// TIA Portal V16 export
// export: Created 2022-02-04T14:40:11.8651462Z, ExportSetting WithDefaults, DisplayName Totally Integrated Automation Portal, DisplayVersion V16 Update 1, DisplayName TIA Portal Version Control Interface, DisplayVersion V16, DisplayName TIA Portal Openness, DisplayVersion V16, DisplayName SINAMICS Startdrive Advanced, DisplayVersion V16 Update 5, DisplayName SINAMICS Startdrive G130, G150, S120, S150, SINAMICS MV, S210, DisplayVersion V16 Update 5, DisplayName SINAMICS Startdrive G110M, G120, G120C, G120D, G120P, G115D, DisplayVersion V16 Update 5, DisplayName STEP 7 Professional, DisplayVersion V16, DisplayName STEP 7 Safety, DisplayVersion V16, DisplayName WinCC Advanced, DisplayVersion V16, DisplayName SIMATIC Visualization Architect, DisplayVersion V16
FUNCTION_BLOCK "Counter_1"   // FB20, LAD
AUTHOR : PSIfunc
VERSION : 0.1
// stored: AutoNumber true, IsIECCheckEnabled false, UDAEnableTagReadback false
   VAR
      SW_GATE_timer : TON;
   END_VAR
BEGIN

REGION Network 1: Запрет счета без движения карусели
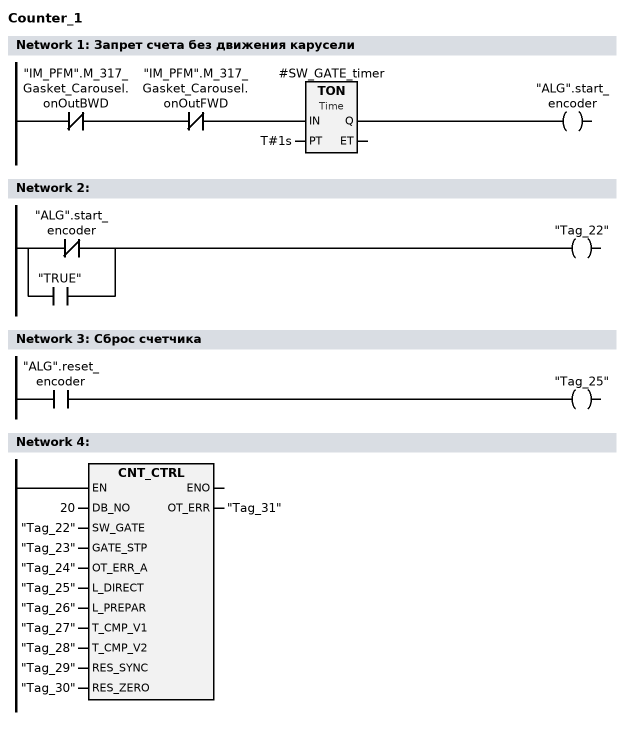
   RUNG wire#powerrail
      I_Contact( "IM_PFM".M_317_Gasket_Carousel.onOutBWD )
      I_Contact( "IM_PFM".M_317_Gasket_Carousel.onOutFWD )
      { S7_Templates := "time_type := Time" } #SW_GATE_timer.TON(pt := T#1s, et =>)
      Coil( "ALG".start_encoder )
   END_RUNG
   // the same network as SCL:
   #SW_GATE_timer.TON(IN := NOT "IM_PFM".M_317_Gasket_Carousel.onOutBWD AND NOT "IM_PFM".M_317_Gasket_Carousel.onOutFWD,
                      PT := T#1s);
   "ALG".start_encoder := #SW_GATE_timer.Q;
END_REGION

REGION Network 2
   RUNG wire#powerrail
      I_Contact( "ALG".start_encoder )
      wire#w1
      Coil( "Tag_22" )
   END_RUNG
   RUNG wire#powerrail
      Contact( "TRUE" )
   END_RUNG wire#w1
   // the same network as SCL:
   "Tag_22" := NOT "ALG".start_encoder OR "TRUE";
END_REGION

REGION Network 3: Сброс счетчика
   RUNG wire#powerrail
      Contact( "ALG".reset_encoder )
      Coil( "Tag_25" )
   END_RUNG
   // the same network as SCL:
   "Tag_25" := "ALG".reset_encoder;
END_REGION

REGION Network 4
   RUNG wire#powerrail
      CNT_CTRL(DB_NO := 20, SW_GATE := "Tag_22", GATE_STP := "Tag_23", OT_ERR_A := "Tag_24", L_DIRECT := "Tag_25", L_PREPAR := "Tag_26", T_CMP_V1 := "Tag_27", T_CMP_V2 := "Tag_28", RES_SYNC := "Tag_29", RES_ZERO := "Tag_30", OT_ERR => "Tag_31")
   END_RUNG
   // the same network as SCL:
   CNT_CTRL(DB_NO := 20,
            SW_GATE := "Tag_22",
            GATE_STP := "Tag_23",
            OT_ERR_A := "Tag_24",
            L_DIRECT := "Tag_25",
            L_PREPAR := "Tag_26",
            T_CMP_V1 := "Tag_27",
            T_CMP_V2 := "Tag_28",
            RES_SYNC := "Tag_29",
            RES_ZERO := "Tag_30",
            OT_ERR => "Tag_31");
END_REGION
END_FUNCTION_BLOCK
